Staubli VAL3: onF7Event.pgx

program onF7Event(bool& x_bSave[])
  local string l_sNew
  local bool l_bUndo
  local num l_nJogVelocity
begin
   // look if the bButton is enable
  if bButton[6]
    //
    //  insert a new entry, it's use a FIFO politic
    //
//    call alreadyExist(l_sNew,l_bUndo)
//    if !l_bUndo and l_sNew!=""
//      call axis:new(l_sNew,nIndex+1)
//      nSelected=nIndex+1
//      call buildList()
//      call refreshStatic()
//      // save it
//      x_bSave=true
//    endIf
    if aioGet(MbAI_b8MotorPow)==1
      //8轴移动速度

      l_nJogVelocity=2
      /////
      aioSet(MbAO_aJogVelo8,l_nJogVelocity)
      aioSet(MbAO_bMoveDir,1)
      aioSet(MbAO_b8Axis,1)
      call use:timerDialog("8轴正向移动...",0)
    else

      if aioGet(MbAI_b8MotorPow)==0
        call use:timerDialog("8轴未上电",1)
        return
      endIf
    endIf
  endIf
end
